FUNCTION_BLOCK FB_BaseMainComponent_HMI EXTENDS FB_BaseComplexElement_HMI IMPLEMENTS ITF_BaseMainComponent_HMI
VAR
	itfBaseMainComponentConnector		: ITF_BaseMainComponent_HMI_Connector;
	refstBaseMainComponentDataHMI		: REFERENCE TO ST_BaseMainComponent_HMI;
END_VAR

END_FUNCTION_BLOCK

(* stored: Version 1.1.0.1
   POU FB_BaseMainComponent_HMI: Id {d9fb61e2-46e3-081a-2db2-ee62cb4cde2f}, SpecialFunc None *)
